PROGRAM MAIN
VAR
END_VAR


// Add and Call Programs to be used 

//	InputMapping();
//	DeviceInputs();
//	Seq1();
//	Safety();
//	MachineStatePackML();
//	DataControl();
//	OutputMapping();
//	DeviceOutputs();
//	EAP_SubscriberMapping();
//	EAP_PublisherMapping();

END_PROGRAM

(* stored: Version 1.1.0.1, ProductVersion 3.1.4024.10
   POU MAIN: Id {4ba25330-7d02-4c90-9be3-142ff1bf6581}, SpecialFunc None *)
